// TwinCAT 3 PLC project PLC
// Title: SARUtills
// Company: Stian Arevoll
// Author: Stian Arevoll
// ProjectVersion: 0.1.2
// ProgramVersion: 3.1.4024.0
// libraries:
//   Tc2_System, * (Beckhoff Automation GmbH)
//   Tc2_Utilities, * (Beckhoff Automation GmbH)
//   Tc3_Module, * (Beckhoff Automation GmbH)
//   TcUnit, * (www.tcunit.org)
// project tree:
//   / PlcTask.TcTTO (not stored)
//   POUs/ FB_Concater.TcPOU, I_Concater.TcIO
//   Tests/ FB_Concater_Test.TcPOU, P_Concater_Tests.TcPOU (not stored)

// ---- POUs/I_Concater.TcIO
INTERFACE I_Concater

METHOD PUBLIC Clear : I_Concater
END_METHOD

METHOD PUBLIC GetString : STRING
END_METHOD

METHOD PUBLIC L : I_Concater
VAR_INPUT
    part : STRING;
END_VAR
END_METHOD

METHOD PUBLIC V : I_Concater
VAR_INPUT
    part : ANY;
END_VAR
END_METHOD

END_INTERFACE

// ---- POUs/FB_Concater.TcPOU
(*
FUNCTION_BLOCK FB_Concater
    VERSION : 1.0

    This function block concatenates strings and variables of various types.
    The concatenated result is stored in an internal buffer which can be retrieved
    using the GetString method. The buffer can be cleared using the Clear method.

    METHODS:
        L(part : STRING) : FB_Concater
            Adds a static string to the buffer.

        V(part : ANY) : FB_Concater
            Adds a variable of any type to the buffer after converting it to a string.

        GetString() : STRING
            Returns the concatenated string stored in the buffer.

        Clear() : FB_Concater
            Clears the buffer.

    PRIVATE METHODS:
        ConvertAnyToString(part : ANY, result : REFERENCE TO STRING) : HRESULT
            Converts a variable of any type to a string.

    EXAMPLE USAGE:
        VAR
            Concater : FB_Concater;
            topic : STRING;
            deviceId : STRING := 'device123';
            sensorType : STRING := 'temperature';
            valueType : STRING := 'reading';
            sensorId : INT := 1;
        END_VAR

        // Building an MQTT topic dynamically
        Concater.Clear().S('home/').V(deviceId).S('/').V(sensorType).S('/').V(sensorId).S('/').V(valueType);
        topic := Concater.GetString();
        // 'topic' will contain: "home/device123/temperature/1/reading"

        // Another example with different values
        Concater.Clear().S('building/').S('office/').V(deviceId).S('/').S('humidity/').V(sensorId).S('/').S('status');
        topic := Concater.GetString();
        // 'topic' will contain: "building/office/device123/humidity/1/status"
*)
FUNCTION_BLOCK FB_Concater IMPLEMENTS I_Concater
VAR
    _buffer : STRING;
    hresult : HRESULT := S_OK;
END_VAR

METHOD PUBLIC Clear : I_Concater
_buffer := '';
Clear := THIS^;
END_METHOD

METHOD PRIVATE ConvertAnyToString : HRESULT
VAR_INPUT
    part : ANY;
    result : REFERENCE TO STRING;
END_VAR
VAR
    pInt : POINTER TO INT;
    pReal : POINTER TO REAL;
    pLReal : POINTER TO LREAL;
    pBool : POINTER TO BOOL;
    pWord : POINTER TO WORD;
    pDWord : POINTER TO DWORD;
    pByte : POINTER TO BYTE;
    pSInt : POINTER TO SINT;
    pUSInt : POINTER TO USINT;
    pDInt : POINTER TO DINT;
    pUDInt : POINTER TO UDINT;
    pLInt : POINTER TO LINT;
    pULInt : POINTER TO ULINT;
	pString	: POINTER TO STRING;
END_VAR

CASE part.TypeClass OF
	__SYSTEM.TYPE_CLASS.TYPE_INT:
		pInt := part.pValue;
		result := INT_TO_STRING(pInt^);
	__SYSTEM.TYPE_CLASS.TYPE_REAL:
		pReal := part.pValue;
		result := REAL_TO_STRING(pReal^);
	__SYSTEM.TYPE_CLASS.TYPE_LREAL:
		pLReal := part.pValue;
		result := LREAL_TO_STRING(pLReal^);
	__SYSTEM.TYPE_CLASS.TYPE_BOOL:
		pBool := part.pValue;
		IF pBool^ THEN
			result := 'TRUE';
		ELSE
			result := 'FALSE';
		END_IF
	__SYSTEM.TYPE_CLASS.TYPE_WORD:
		pWord := part.pValue;
		result := WORD_TO_STRING(pWord^);
	__SYSTEM.TYPE_CLASS.TYPE_DWORD:
		pDWord := part.pValue;
		result := DWORD_TO_STRING(pDWord^);
	__SYSTEM.TYPE_CLASS.TYPE_BYTE:
		pByte := part.pValue;
		result := BYTE_TO_STRING(pByte^);
	__SYSTEM.TYPE_CLASS.TYPE_SINT:
		pSInt := part.pValue;
		result := SINT_TO_STRING(pSInt^);
	__SYSTEM.TYPE_CLASS.TYPE_USINT:
		pUSInt := part.pValue;
		result := USINT_TO_STRING(pUSInt^);
	__SYSTEM.TYPE_CLASS.TYPE_DINT:
		pDInt := part.pValue;
		result := DINT_TO_STRING(pDInt^);
	__SYSTEM.TYPE_CLASS.TYPE_UDINT:
		pUDInt := part.pValue;
		result := UDINT_TO_STRING(pUDInt^);
	__SYSTEM.TYPE_CLASS.TYPE_LINT:
		pLInt := part.pValue;
		result := LINT_TO_STRING(pLInt^);
	__SYSTEM.TYPE_CLASS.TYPE_ULINT:
		pULInt := part.pValue;
		result := ULINT_TO_STRING(pULInt^);
	__SYSTEM.TYPE_CLASS.TYPE_STRING:
		pString := part.pValue;
		result := pString^; 
	ELSE
		ConvertAnyToString := E_FAIL;
		RETURN;
END_CASE
ConvertAnyToString := S_OK;
END_METHOD

METHOD PUBLIC GetString : STRING
GetString := _buffer;
END_METHOD

METHOD PUBLIC L : I_Concater
VAR_INPUT
    part : STRING;
END_VAR
L := THIS^.V(part);
END_METHOD

METHOD PUBLIC V : I_Concater
VAR_INPUT
    part : ANY;
END_VAR
VAR
    strPart : STRING;
END_VAR
hresult := ConvertAnyToString(part, strPart);

IF FAILED(hresult) THEN
	_buffer := 'Error: Unsupported type';
	V := THIS^;
	RETURN;
END_IF

CONCAT2(ADR(_buffer), ADR(strPart), ADR(_buffer), SIZEOF(_buffer));
V := THIS^;
END_METHOD

END_FUNCTION_BLOCK

// ---- Tests/FB_Concater_Test.TcPOU
FUNCTION_BLOCK FB_Concater_Test EXTENDS TcUnit.FB_TestSuite
VAR
	fbConcater : FB_Concater;
	
    stringResult : STRING;
    myInt : INT := 123;
    myReal : REAL := 45.67;
    myLReal : LREAL := 12345.6789;
    myBool : BOOL := TRUE;
    myWord : WORD := 16#ABCD;
    myString : STRING := 'example';
    myDInt : DINT := -456;
    myUDInt : UDINT := 789;
    myLInt : LINT := -123456789;
    myULInt : ULINT := 123456789;
END_VAR

TEST('TestClearMethod');
    fbConcater.L('test');
    fbConcater.Clear();
    stringResult := fbConcater.GetString();
	AssertEquals_STRING('', stringResult, 'Test of Clear method failed');
TEST_FINISHED();

TEST('TestGetStringMethod');
	fbConcater.Clear().L('test');
    stringResult := fbConcater.GetString();
    AssertEquals_STRING('test', stringResult, 'Test of GetString method failed');
TEST_FINISHED();

TEST('TestConcatStaticStrings');
    fbConcater.Clear().L('my/').L('static/').L('strings');
    stringResult := fbConcater.GetString();
    AssertEquals_STRING('my/static/strings', stringResult, 'Test with static strings failed');
TEST_FINISHED();

TEST('TestConcatInteger');
    fbConcater.Clear().V(myInt).L('/').V(myDInt).L('/').V(myUDInt);
    stringResult := fbConcater.GetString();
    AssertEquals_STRING('123/-456/789', stringResult, 'Test with integers failed');
TEST_FINISHED();

TEST('TestConcatReal');
    fbConcater.Clear().V(myReal);
    stringResult := fbConcater.GetString();
    AssertEquals_STRING('45.67', stringResult, 'Test with real number failed');
TEST_FINISHED();

TEST('TestConcatLReal');
    fbConcater.Clear().V(myLReal);
    stringResult := fbConcater.GetString();
    AssertEquals_STRING('12345.6789', stringResult, 'Test with LREAL failed');
TEST_FINISHED();

TEST('TestConcatBool');
    fbConcater.Clear().V(myBool);
    stringResult := fbConcater.GetString();
    AssertEquals_STRING('TRUE', stringResult, 'Test with boolean value TRUE failed');

    fbConcater.Clear().L('FALSE');
    stringResult := fbConcater.GetString();
    AssertEquals_STRING('FALSE', stringResult, 'Test with boolean value FALSE failed');
TEST_FINISHED();

TEST('TestConcatWord');
    fbConcater.Clear().V(myWord);
    stringResult := fbConcater.GetString();
    AssertEquals_STRING('43981', stringResult, 'Test with WORD failed'); // 16#ABCD = 43981
TEST_FINISHED();

TEST('TestConcatLIntAndULInt');
    fbConcater.Clear().V(myLInt).L('/').V(myULInt);
    stringResult := fbConcater.GetString();
    AssertEquals_STRING('-123456789/123456789', stringResult, 'Test with LINT and ULINT failed');
TEST_FINISHED();

TEST('TestMixedConcat');
    fbConcater.Clear().V(myInt).L('/').V(myReal).L('/').V(myBool).L('/').V(myWord).L('/').V(myString);
    stringResult := fbConcater.GetString();
    AssertEquals_STRING('123/45.67/TRUE/43981/example', stringResult, 'Test with mixed types failed');
TEST_FINISHED();

METHOD Tests : BOOL
(*

TEST('TestClearMethod');
    fbConcater.L('test');
    fbConcater.Clear();
    stringResult := fbConcater.GetString();
	AssertEquals_STRING('', stringResult, 'Test of Clear method failed');
TEST_FINISHED();

TEST('TestGetStringMethod');
	fbConcater.Clear().L('test');
    stringResult := fbConcater.GetString();
    AssertEquals_STRING('test', stringResult, 'Test of GetString method failed');
TEST_FINISHED();

TEST('TestConcatStaticStrings');
    fbConcater.Clear().L('my/').L('static/').L('strings');
    stringResult := fbConcater.GetString();
    AssertEquals_STRING('my/static/strings', stringResult, 'Test with static strings failed');
TEST_FINISHED();

TEST('TestConcatInteger');
    fbConcater.Clear().V(myInt).L('/').V(myDInt).L('/').V(myUDInt);
    stringResult := fbConcater.GetString();
    AssertEquals_STRING('123/-456/789', stringResult, 'Test with integers failed');
TEST_FINISHED();

TEST('TestConcatReal');
    fbConcater.Clear().V(myReal);
    stringResult := fbConcater.GetString();
    AssertEquals_STRING('45.67', stringResult, 'Test with real number failed');
TEST_FINISHED();

TEST('TestConcatLReal');
    fbConcater.Clear().V(myLReal);
    stringResult := fbConcater.GetString();
    AssertEquals_STRING('12345.6789', stringResult, 'Test with LREAL failed');
TEST_FINISHED();

TEST('TestConcatBool');
    fbConcater.Clear().V(myBool);
    stringResult := fbConcater.GetString();
    AssertEquals_STRING('TRUE', stringResult, 'Test with boolean value TRUE failed');

    fbConcater.Clear().L('FALSE');
    stringResult := fbConcater.GetString();
    AssertEquals_STRING('FALSE', stringResult, 'Test with boolean value FALSE failed');
TEST_FINISHED();

TEST('TestConcatWord');
    fbConcater.Clear().V(myWord);
    stringResult := fbConcater.GetString();
    AssertEquals_STRING('43981', stringResult, 'Test with WORD failed'); // 16#ABCD = 43981
TEST_FINISHED();

TEST('TestConcatLIntAndULInt');
    fbConcater.Clear().V(myLInt).L('/').V(myULInt);
    stringResult := fbConcater.GetString();
    AssertEquals_STRING('-123456789/123456789', stringResult, 'Test with LINT and ULINT failed');
TEST_FINISHED();

TEST('TestMixedConcat');
    fbConcater.Clear().V(myInt).L('/').V(myReal).L('/').V(myBool).L('/').V(myWord).L('/').V(myString);
    stringResult := fbConcater.GetString();
    AssertEquals_STRING('123/45.67/TRUE/43981/example', stringResult, 'Test with mixed types failed');
TEST_FINISHED();

*)
END_METHOD

END_FUNCTION_BLOCK
